PROGRAM PRG_SystemControlMachineWork
VAR
END_VAR

IF (PRG_SystemControlMachineInit.bFirstCycle) THEN
	GVL_SystemVariable.fbLogger ();
	GVL_SystemVariable.fbMachineControl ();
END_IF

END_PROGRAM

(* stored: Version 1.1.0.1
   POU PRG_SystemControlMachineWork: Id {79612be6-fc24-0aa2-1eaf-ef9f7362db8a}, SpecialFunc None *)
